(* PLC project v0.6.02_RefactorGateAndTest.project, CODESYS CODESYS V3.5 SP19 Patch 1 *)
(* stored: creationDateTime 2026-08-14T10:10:49.365026, modificationDateTime 2026-08-14T10:10:49.365026 *)

(* ═══════════════════════════════════════════════════════════════ 💓 FB_Diag_IhmHeartbeat — Surveillance bidirectionnelle IHM↔PLC ─────────────────────────────────────────────────────────────── 📄 Doc : DOC/AF/AF_Partie-07_Interface_IHM_v2.0.md (mise à jour Heartbeat requise) 🧩 Brique réduite : surveille le toggle IHM, génère le toggle PLC et expose un diagnostic. Ne produit ni SafeStop ni PowerCutOff. 🛡️ Les FB_Safety_Winch / FB_Safety_Translation restent propriétaires de leurs réactions métier. ═══════════════════════════════════════════════════════════════ *)
FUNCTION_BLOCK FB_Diag_IhmHeartbeat
  VAR_INPUT
    Enable : BOOL;  (* Active la surveillance ; FALSE = IHM non valide *)
    TglHeartbeatIhm : BOOL;  (* Toggle IHM, inversion attendue toutes les 500 ms *)
    IhmTimeout : TIME := TIME#2s0ms;  (* Absence maximale de front IHM *)
    PlcTogglePeriod : TIME := TIME#500ms;  (* Période du clignotant PLC *)
  END_VAR
  VAR_OUTPUT
    HeartbeatIhmOk : BOOL;  (* TRUE après front IHM post-boot et avant timeout *)
    HeartbeatIhmTimeout : BOOL;  (* TRUE = aucun front IHM depuis IhmTimeout *)
    TglHeartbeatPlc : BOOL;  (* Clignotant PLC à superviser côté IHM *)
    TimeSinceIhmEdge : TIME;  (* Diagnostic : temps depuis le dernier front IHM *)
  END_VAR
  VAR
    LastIhmToggle : BOOL;
    IhmEdgeSeen : BOOL;  (* Interdit de valider une valeur RETAIN au boot *)
    IhmEdgeDetected : BOOL;
    IhmTimeoutTon : TON;
    PlcToggleTon : TON;
  END_VAR

            

// === IMPLEMENTATION ===

// 🛑 Sans Enable, aucune valeur mémorisée ne peut déclarer l'IHM valide.
IF NOT Enable THEN
    HeartbeatIhmOk := FALSE;
    HeartbeatIhmTimeout := TRUE;
    TglHeartbeatPlc := FALSE;
    TimeSinceIhmEdge := T#0s;
    LastIhmToggle := TglHeartbeatIhm;
    IhmEdgeSeen := FALSE;
    IhmTimeoutTon(IN := FALSE, PT := IhmTimeout);
    PlcToggleTon(IN := FALSE, PT := PlcTogglePeriod);
    RETURN;
END_IF;

// 📥 Front par comparaison : l'IHM écrit un BOOL toggle, pas une impulsion courte.
IhmEdgeDetected := (TglHeartbeatIhm <> LastIhmToggle);
LastIhmToggle := TglHeartbeatIhm;
IF IhmEdgeDetected THEN
    IhmEdgeSeen := TRUE;
END_IF;

// ⏱️ Le timer repart à chaque front. Au boot, il atteint le timeout au bout de IhmTimeout.
// HeartbeatIhmOk reste TRUE tant que le timeout n'est pas expiré (boot propre sans alarme au scan 1).
IhmTimeoutTon(IN := NOT IhmEdgeDetected, PT := IhmTimeout);
TimeSinceIhmEdge := IhmTimeoutTon.ET;
HeartbeatIhmTimeout := IhmTimeoutTon.Q;
HeartbeatIhmOk := NOT HeartbeatIhmTimeout;

// 💡 Clignotant PLC indépendant : information de vie pour l'IHM, jamais signal Safety autonome.
PlcToggleTon(IN := NOT PlcToggleTon.Q, PT := PlcTogglePeriod);
IF PlcToggleTon.Q THEN
    TglHeartbeatPlc := NOT TglHeartbeatPlc;
END_IF;

          
END_FUNCTION_BLOCK
